(* Logix 5000 project; controller SX_V040001_C001 vendor 1 type 14 code 77 rev 16.22; software revision 16.04; part 16 of 35 *)
(* tags used below, declared in another part *)
   ALL_KINDS : INT[90];
   DRIVE : INT[32];
   G_AOutput : DINT[8];
   G_DInput : DINT[3];
   G_DOutput : DINT[3];
   NOTDOS : INT[6];
   PARAMETER : INT[501];
   T_CONTR_CLFA_ACLFA : TIMER;
   T_CURRENT_AUTO : TIMER;
   T_CURRENT_CL : TIMER;
   T_DELAY_SLOW_FAST : TIMER;
   T_DELAY_SOFTSTART : TIMER;
   T_DRIVE_START_WARN : TIMER;
(* MainProgram, continued *)

ROUTINE MainDrive2Motors   (* ladder *)
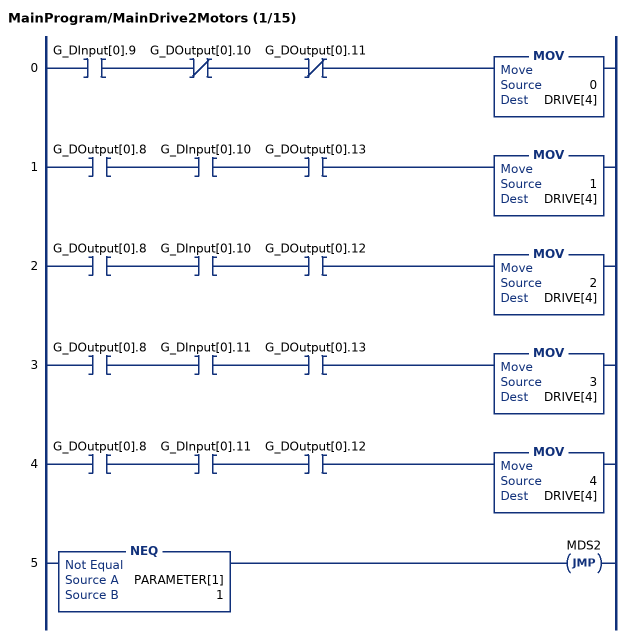
   0: XIC(G_DInput[0].9)XIO(G_DOutput[0].10)XIO(G_DOutput[0].11)MOV(0,DRIVE[4]);
   1: XIC(G_DOutput[0].8)XIC(G_DInput[0].10)XIC(G_DOutput[0].13)MOV(1,DRIVE[4]);
   2: XIC(G_DOutput[0].8)XIC(G_DInput[0].10)XIC(G_DOutput[0].12)MOV(2,DRIVE[4]);
   3: XIC(G_DOutput[0].8)XIC(G_DInput[0].11)XIC(G_DOutput[0].13)MOV(3,DRIVE[4]);
   4: XIC(G_DOutput[0].8)XIC(G_DInput[0].11)XIC(G_DOutput[0].12)MOV(4,DRIVE[4]);
   5: NEQ(PARAMETER[1],1)JMP(MDS2);
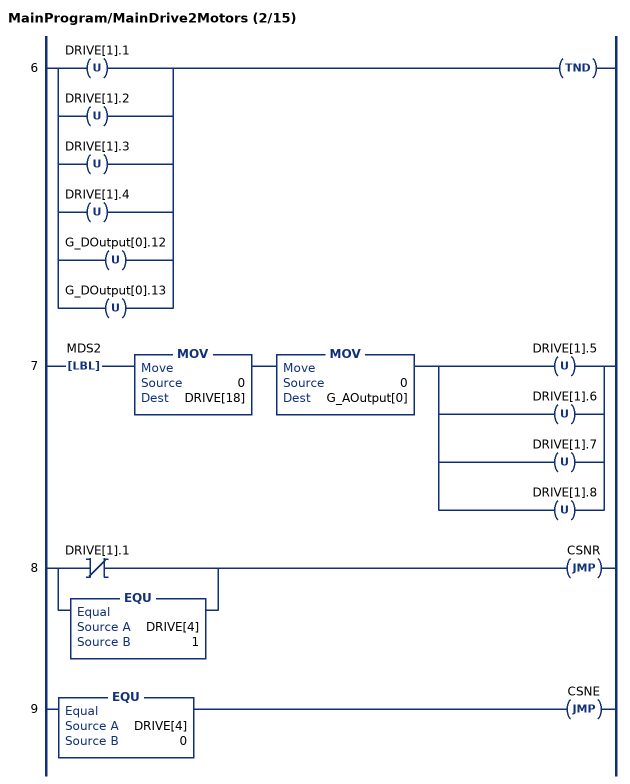
   6: [OTU(DRIVE[1].1) ,OTU(DRIVE[1].2) ,OTU(DRIVE[1].3) ,OTU(DRIVE[1].4) ,OTU(G_DOutput[0].12) ,OTU(G_DOutput[0].13) ]TND();
   7: LBL(MDS2)MOV(0,DRIVE[18])MOV(0,G_AOutput[0])[OTU(DRIVE[1].5) ,OTU(DRIVE[1].6) ,OTU(DRIVE[1].7) ,OTU(DRIVE[1].8) ];
   8: [XIO(DRIVE[1].1) ,EQU(DRIVE[4],1) ]JMP(CSNR);
   9: EQU(DRIVE[4],0)JMP(CSNE);
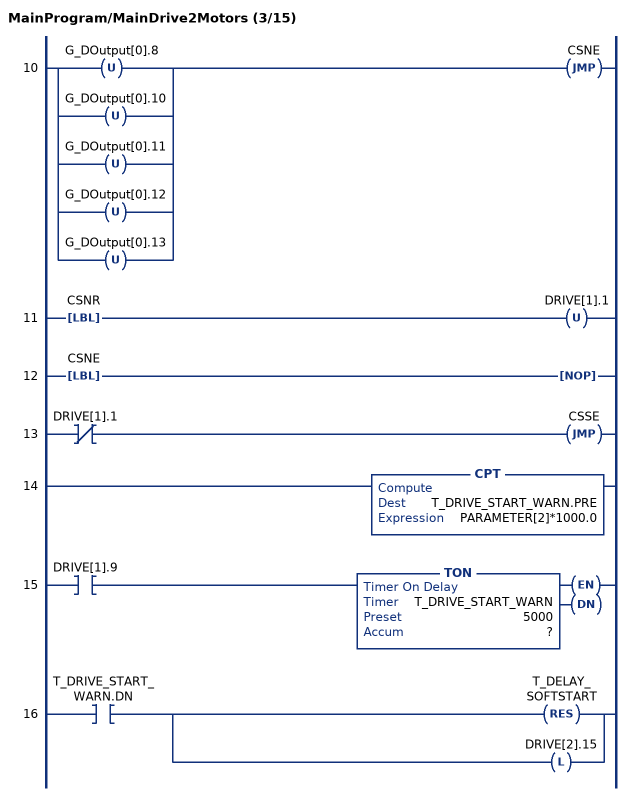
   10: [OTU(G_DOutput[0].8) ,OTU(G_DOutput[0].10) ,OTU(G_DOutput[0].11) ,OTU(G_DOutput[0].12) ,OTU(G_DOutput[0].13) ]JMP(CSNE);
   11: LBL(CSNR)OTU(DRIVE[1].1);
   12: LBL(CSNE)NOP();
   13: XIO(DRIVE[1].1)JMP(CSSE);
   14: CPT(T_DRIVE_START_WARN.PRE,PARAMETER[2]*1000.0);
   15: XIC(DRIVE[1].9)TON(T_DRIVE_START_WARN,?,?);
   16: XIC(T_DRIVE_START_WARN.DN)[RES(T_DELAY_SOFTSTART) ,OTL(DRIVE[2].15) ];
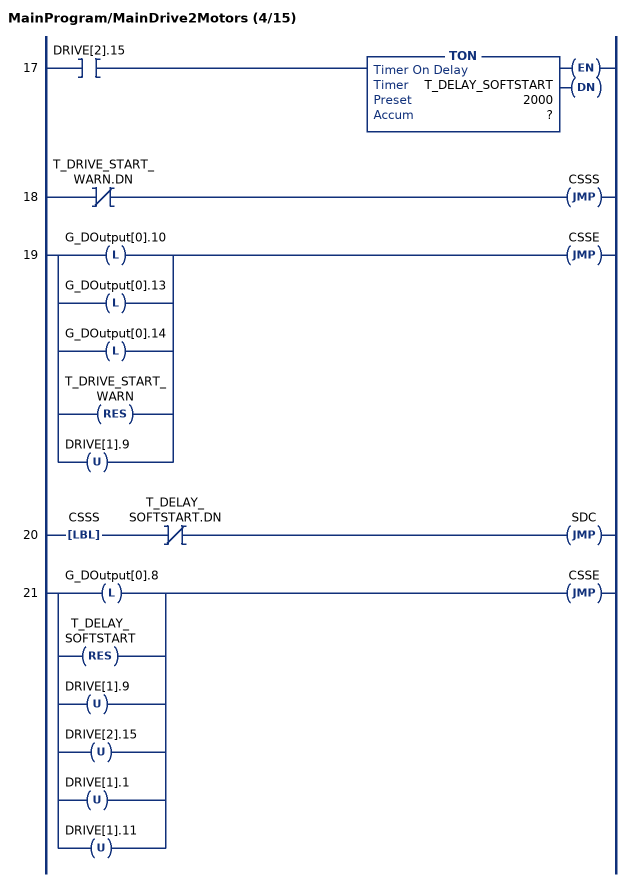
   17: XIC(DRIVE[2].15)TON(T_DELAY_SOFTSTART,?,?);
   18: XIO(T_DRIVE_START_WARN.DN)JMP(CSSS);
   19: [OTL(G_DOutput[0].10) ,OTL(G_DOutput[0].13) ,OTL(G_DOutput[0].14) ,RES(T_DRIVE_START_WARN) ,OTU(DRIVE[1].9) ]JMP(CSSE);
   20: LBL(CSSS)XIO(T_DELAY_SOFTSTART.DN)JMP(SDC);
   21: [OTL(G_DOutput[0].8) ,RES(T_DELAY_SOFTSTART) ,OTU(DRIVE[1].9) ,OTU(DRIVE[2].15) ,OTU(DRIVE[1].1) ,OTU(DRIVE[1].11) ]JMP(CSSE);
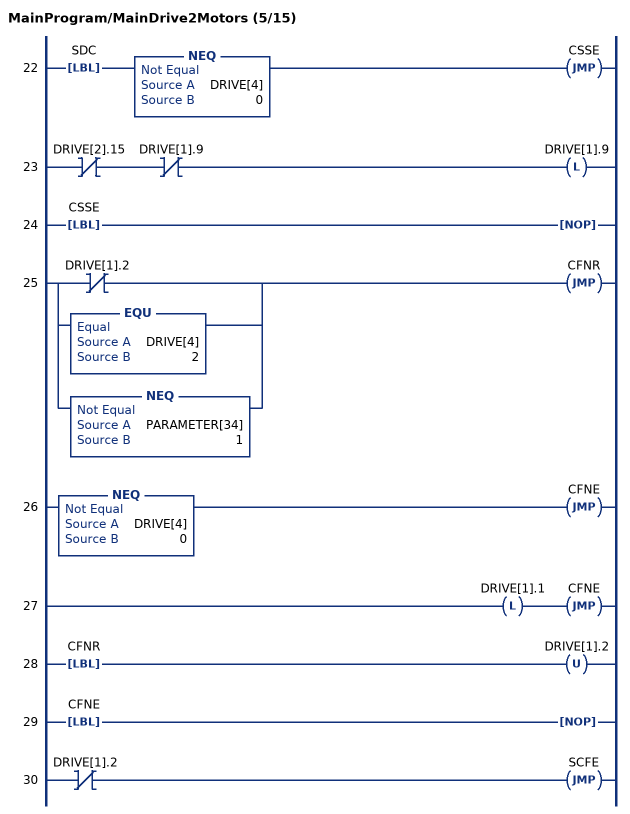
   22: LBL(SDC)NEQ(DRIVE[4],0)JMP(CSSE);
   23: XIO(DRIVE[2].15)XIO(DRIVE[1].9)OTL(DRIVE[1].9);
   24: LBL(CSSE)NOP();
   25: [XIO(DRIVE[1].2) ,EQU(DRIVE[4],2) ,NEQ(PARAMETER[34],1) ]JMP(CFNR);
   26: NEQ(DRIVE[4],0)JMP(CFNE);
   27: OTL(DRIVE[1].1)JMP(CFNE);
   28: LBL(CFNR)OTU(DRIVE[1].2);
   29: LBL(CFNE)NOP();
   30: XIO(DRIVE[1].2)JMP(SCFE);
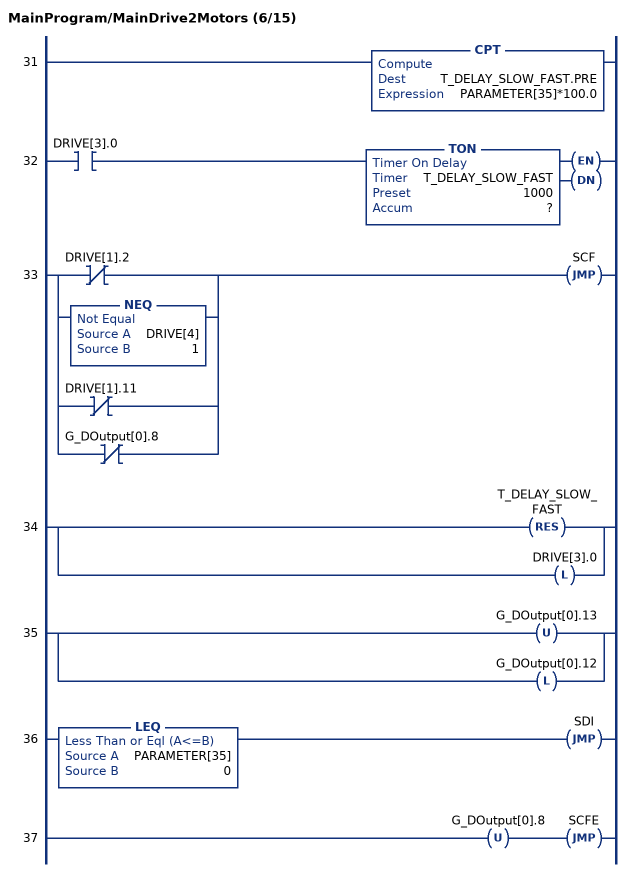
   31: CPT(T_DELAY_SLOW_FAST.PRE,PARAMETER[35]*100.0);
   32: XIC(DRIVE[3].0)TON(T_DELAY_SLOW_FAST,?,?);
   33: [XIO(DRIVE[1].2) ,NEQ(DRIVE[4],1) ,XIO(DRIVE[1].11) ,XIO(G_DOutput[0].8) ]JMP(SCF);
   34: [RES(T_DELAY_SLOW_FAST) ,OTL(DRIVE[3].0) ];
   35: [OTU(G_DOutput[0].13) ,OTL(G_DOutput[0].12) ];
   36: LEQ(PARAMETER[35],0)JMP(SDI);
   37: OTU(G_DOutput[0].8)JMP(SCFE);
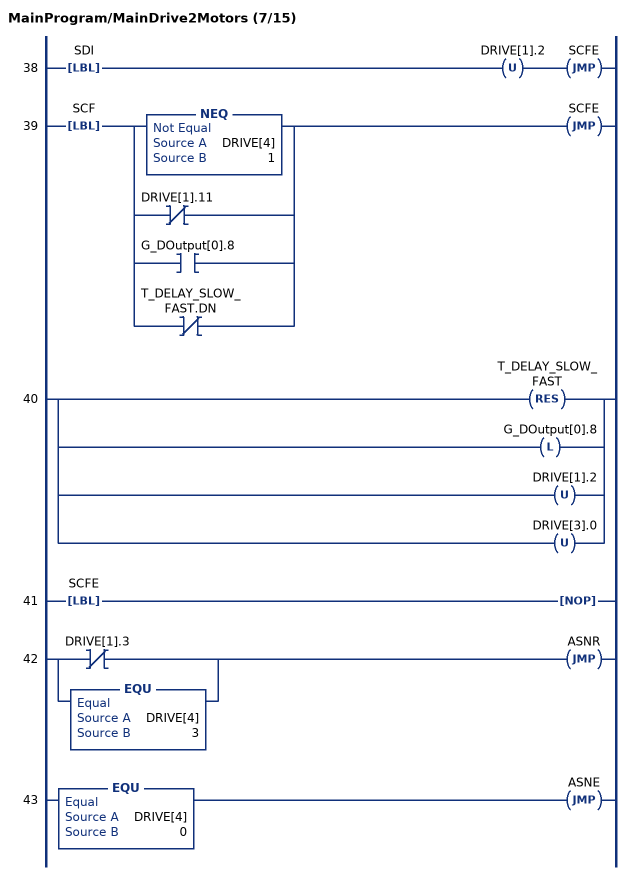
   38: LBL(SDI)OTU(DRIVE[1].2)JMP(SCFE);
   39: LBL(SCF)[NEQ(DRIVE[4],1) ,XIO(DRIVE[1].11) ,XIC(G_DOutput[0].8) ,XIO(T_DELAY_SLOW_FAST.DN) ]JMP(SCFE);
   40: [RES(T_DELAY_SLOW_FAST) ,OTL(G_DOutput[0].8) ,OTU(DRIVE[1].2) ,OTU(DRIVE[3].0) ];
   41: LBL(SCFE)NOP();
   42: [XIO(DRIVE[1].3) ,EQU(DRIVE[4],3) ]JMP(ASNR);
   43: EQU(DRIVE[4],0)JMP(ASNE);
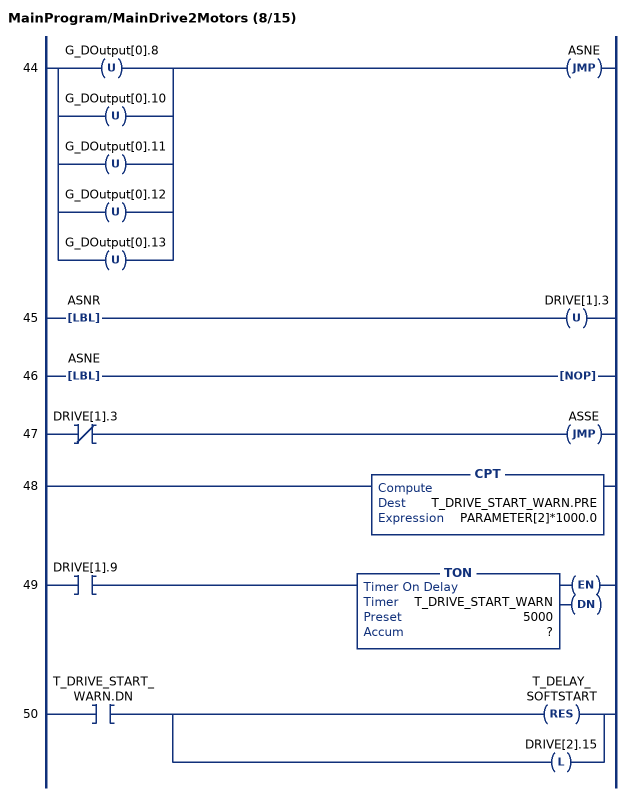
   44: [OTU(G_DOutput[0].8) ,OTU(G_DOutput[0].10) ,OTU(G_DOutput[0].11) ,OTU(G_DOutput[0].12) ,OTU(G_DOutput[0].13) ]JMP(ASNE);
   45: LBL(ASNR)OTU(DRIVE[1].3);
   46: LBL(ASNE)NOP();
   47: XIO(DRIVE[1].3)JMP(ASSE);
   48: CPT(T_DRIVE_START_WARN.PRE,PARAMETER[2]*1000.0);
   49: XIC(DRIVE[1].9)TON(T_DRIVE_START_WARN,?,?);
   50: XIC(T_DRIVE_START_WARN.DN)[RES(T_DELAY_SOFTSTART) ,OTL(DRIVE[2].15) ];
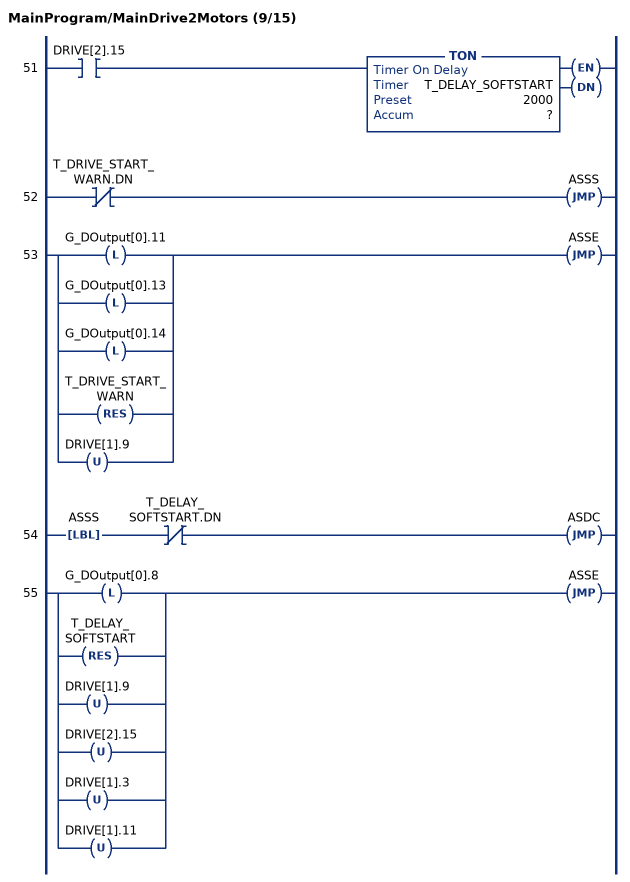
   51: XIC(DRIVE[2].15)TON(T_DELAY_SOFTSTART,?,?);
   52: XIO(T_DRIVE_START_WARN.DN)JMP(ASSS);
   53: [OTL(G_DOutput[0].11) ,OTL(G_DOutput[0].13) ,OTL(G_DOutput[0].14) ,RES(T_DRIVE_START_WARN) ,OTU(DRIVE[1].9) ]JMP(ASSE);
   54: LBL(ASSS)XIO(T_DELAY_SOFTSTART.DN)JMP(ASDC);
   55: [OTL(G_DOutput[0].8) ,RES(T_DELAY_SOFTSTART) ,OTU(DRIVE[1].9) ,OTU(DRIVE[2].15) ,OTU(DRIVE[1].3) ,OTU(DRIVE[1].11) ]JMP(ASSE);
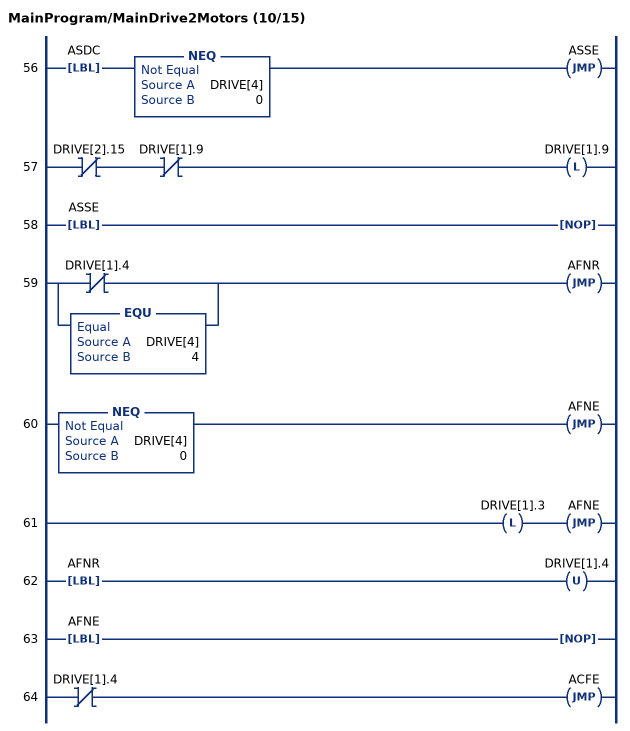
   56: LBL(ASDC)NEQ(DRIVE[4],0)JMP(ASSE);
   57: XIO(DRIVE[2].15)XIO(DRIVE[1].9)OTL(DRIVE[1].9);
   58: LBL(ASSE)NOP();
   59: [XIO(DRIVE[1].4) ,EQU(DRIVE[4],4) ]JMP(AFNR);
   60: NEQ(DRIVE[4],0)JMP(AFNE);
   61: OTL(DRIVE[1].3)JMP(AFNE);
   62: LBL(AFNR)OTU(DRIVE[1].4);
   63: LBL(AFNE)NOP();
   64: XIO(DRIVE[1].4)JMP(ACFE);
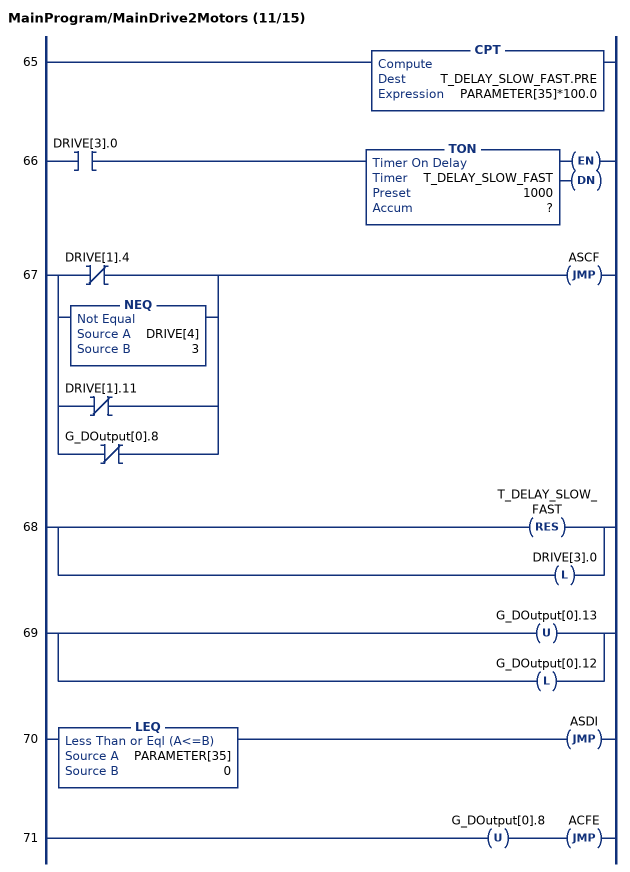
   65: CPT(T_DELAY_SLOW_FAST.PRE,PARAMETER[35]*100.0);
   66: XIC(DRIVE[3].0)TON(T_DELAY_SLOW_FAST,?,?);
   67: [XIO(DRIVE[1].4) ,NEQ(DRIVE[4],3) ,XIO(DRIVE[1].11) ,XIO(G_DOutput[0].8) ]JMP(ASCF);
   68: [RES(T_DELAY_SLOW_FAST) ,OTL(DRIVE[3].0) ];
   69: [OTU(G_DOutput[0].13) ,OTL(G_DOutput[0].12) ];
   70: LEQ(PARAMETER[35],0)JMP(ASDI);
   71: OTU(G_DOutput[0].8)JMP(ACFE);
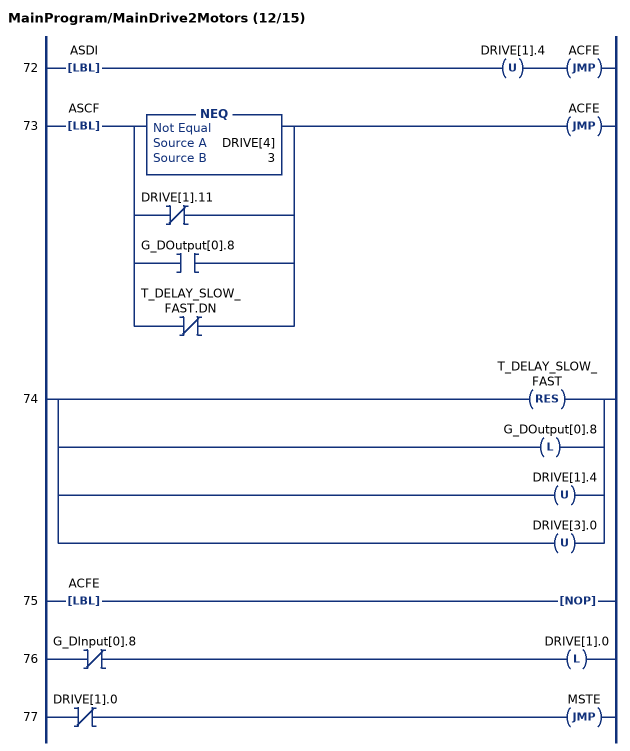
   72: LBL(ASDI)OTU(DRIVE[1].4)JMP(ACFE);
   73: LBL(ASCF)[NEQ(DRIVE[4],3) ,XIO(DRIVE[1].11) ,XIC(G_DOutput[0].8) ,XIO(T_DELAY_SLOW_FAST.DN) ]JMP(ACFE);
   74: [RES(T_DELAY_SLOW_FAST) ,OTL(G_DOutput[0].8) ,OTU(DRIVE[1].4) ,OTU(DRIVE[3].0) ];
   75: LBL(ACFE)NOP();
   76: XIO(G_DInput[0].8)OTL(DRIVE[1].0);
   77: XIO(DRIVE[1].0)JMP(MSTE);
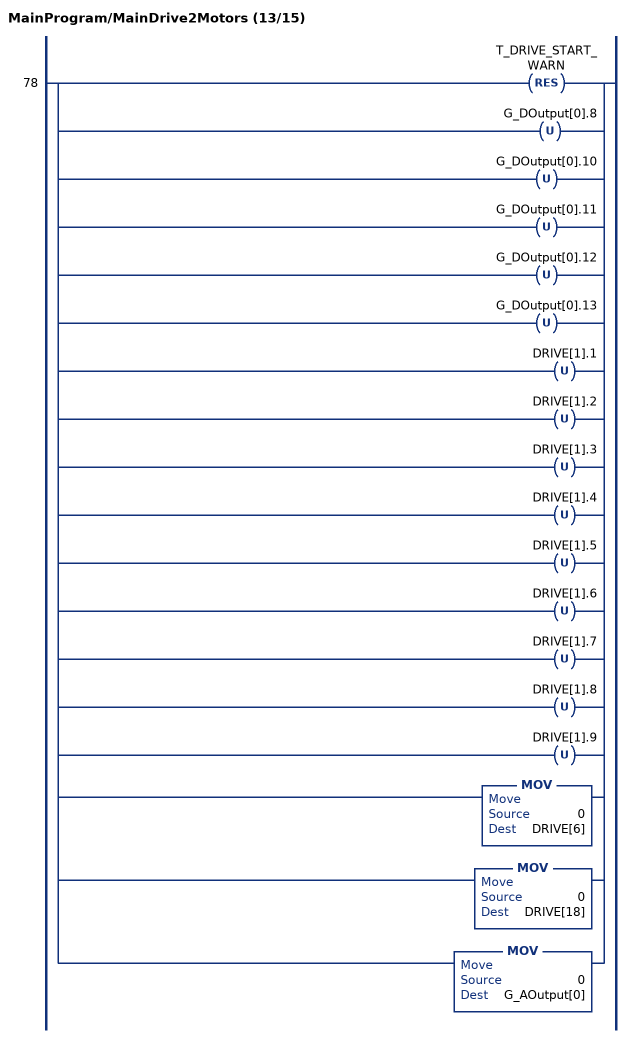
   78: [RES(T_DRIVE_START_WARN) ,OTU(G_DOutput[0].8) ,OTU(G_DOutput[0].10) ,OTU(G_DOutput[0].11) ,OTU(G_DOutput[0].12) ,OTU(G_DOutput[0].13) ,OTU(DRIVE[1].1) ,OTU(DRIVE[1].2) ,OTU(DRIVE[1].3) ,OTU(DRIVE[1].4) ,OTU(DRIVE[1].5) ,OTU(DRIVE[1].6) ,OTU(DRIVE[1].7) ,OTU(DRIVE[1].8) ,OTU(DRIVE[1].9) ,MOV(0,DRIVE[6]) ,MOV(0,DRIVE[18]) ,MOV(0,G_AOutput[0]) ];
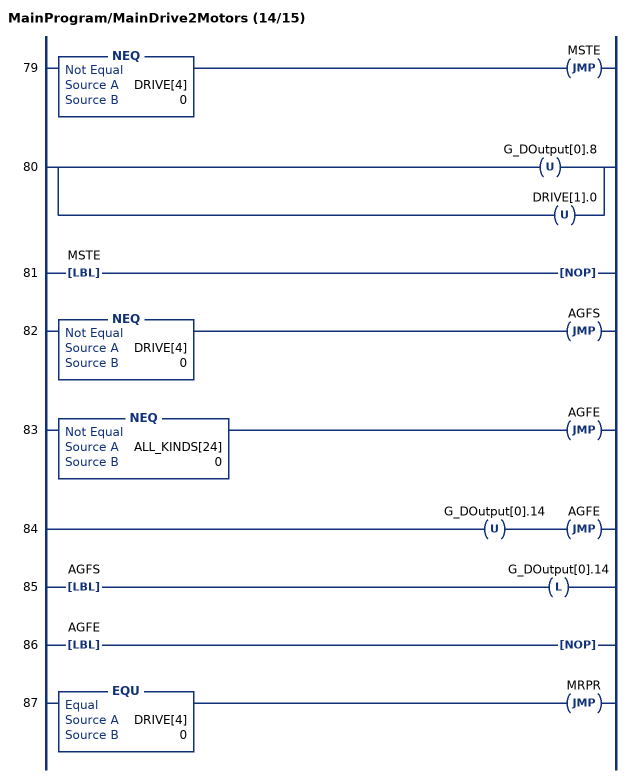
   79: NEQ(DRIVE[4],0)JMP(MSTE);
   80: [OTU(G_DOutput[0].8) ,OTU(DRIVE[1].0) ];
   81: LBL(MSTE)NOP();
   82: NEQ(DRIVE[4],0)JMP(AGFS);
   83: NEQ(ALL_KINDS[24],0)JMP(AGFE);
   84: OTU(G_DOutput[0].14)JMP(AGFE);
   85: LBL(AGFS)OTL(G_DOutput[0].14);
   86: LBL(AGFE)NOP();
   87: EQU(DRIVE[4],0)JMP(MRPR);
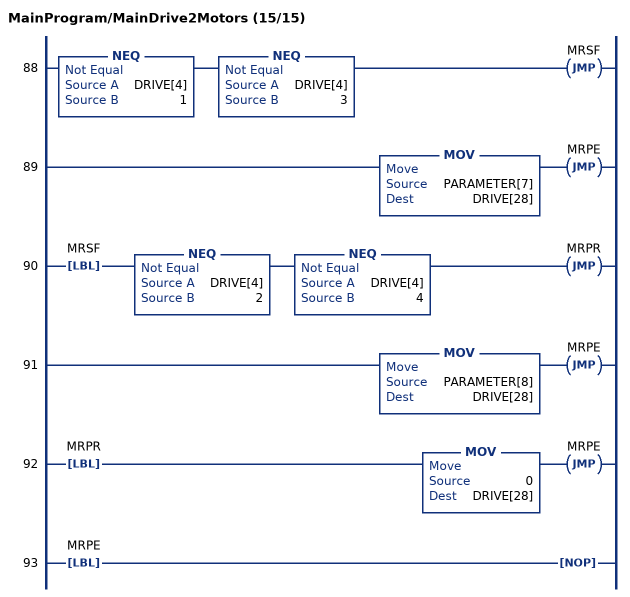
   88: NEQ(DRIVE[4],1)NEQ(DRIVE[4],3)JMP(MRSF);
   89: MOV(PARAMETER[7],DRIVE[28])JMP(MRPE);
   90: LBL(MRSF)NEQ(DRIVE[4],2)NEQ(DRIVE[4],4)JMP(MRPR);
   91: MOV(PARAMETER[8],DRIVE[28])JMP(MRPE);
   92: LBL(MRPR)MOV(0,DRIVE[28])JMP(MRPE);
   93: LBL(MRPE)NOP();
END_ROUTINE

ROUTINE MainDriveCurrent   (* ladder *)
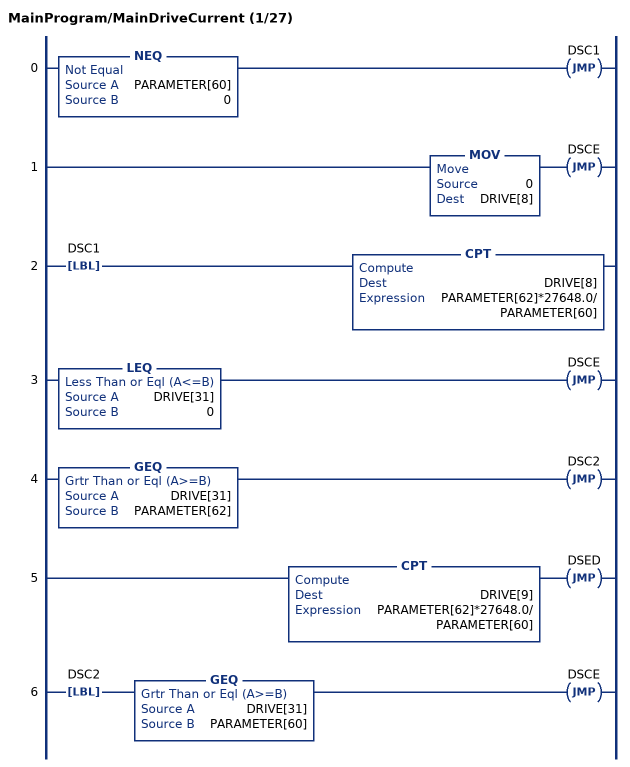
   0: NEQ(PARAMETER[60],0)JMP(DSC1);
   1: MOV(0,DRIVE[8])JMP(DSCE);
   2: LBL(DSC1)CPT(DRIVE[8],PARAMETER[62]*27648.0/PARAMETER[60]);
   3: LEQ(DRIVE[31],0)JMP(DSCE);
   4: GEQ(DRIVE[31],PARAMETER[62])JMP(DSC2);
   5: CPT(DRIVE[9],PARAMETER[62]*27648.0/PARAMETER[60])JMP(DSED);
   6: LBL(DSC2)GEQ(DRIVE[31],PARAMETER[60])JMP(DSCE);
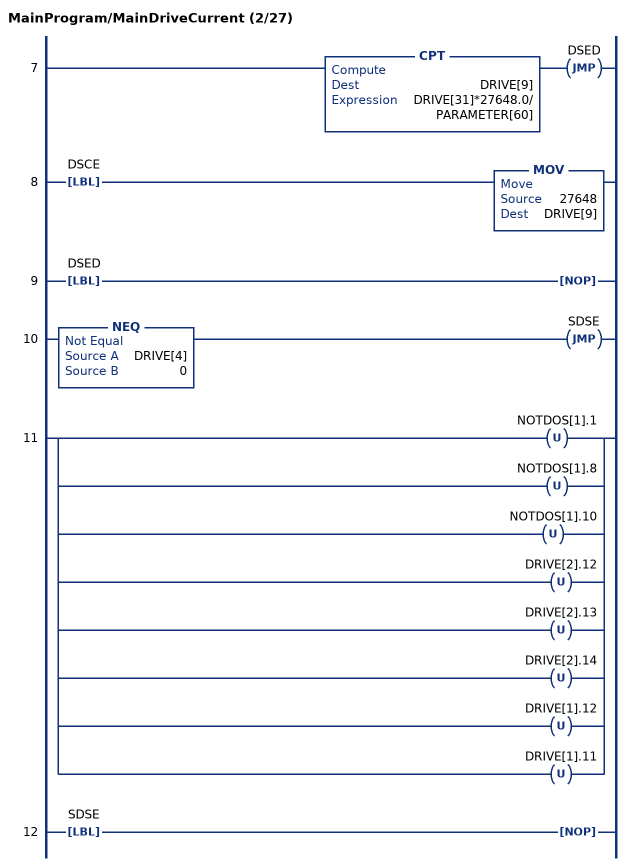
   7: CPT(DRIVE[9],DRIVE[31]*27648.0/PARAMETER[60])JMP(DSED);
   8: LBL(DSCE)MOV(27648,DRIVE[9]);
   9: LBL(DSED)NOP();
   10: NEQ(DRIVE[4],0)JMP(SDSE);
   11: [OTU(NOTDOS[1].1) ,OTU(NOTDOS[1].8) ,OTU(NOTDOS[1].10) ,OTU(DRIVE[2].12) ,OTU(DRIVE[2].13) ,OTU(DRIVE[2].14) ,OTU(DRIVE[1].12) ,OTU(DRIVE[1].11) ];
   12: LBL(SDSE)NOP();
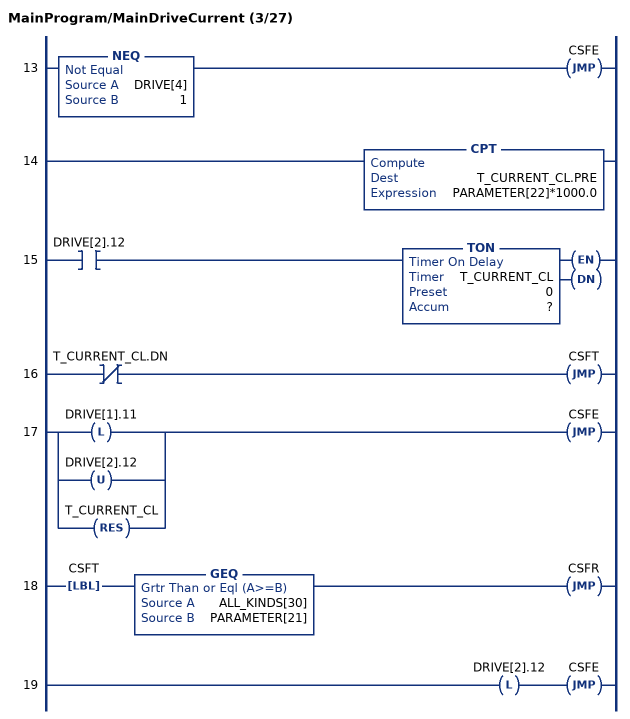
   13: NEQ(DRIVE[4],1)JMP(CSFE);
   14: CPT(T_CURRENT_CL.PRE,PARAMETER[22]*1000.0);
   15: XIC(DRIVE[2].12)TON(T_CURRENT_CL,?,?);
   16: XIO(T_CURRENT_CL.DN)JMP(CSFT);
   17: [OTL(DRIVE[1].11) ,OTU(DRIVE[2].12) ,RES(T_CURRENT_CL) ]JMP(CSFE);
   18: LBL(CSFT)GEQ(ALL_KINDS[30],PARAMETER[21])JMP(CSFR);
   19: OTL(DRIVE[2].12)JMP(CSFE);
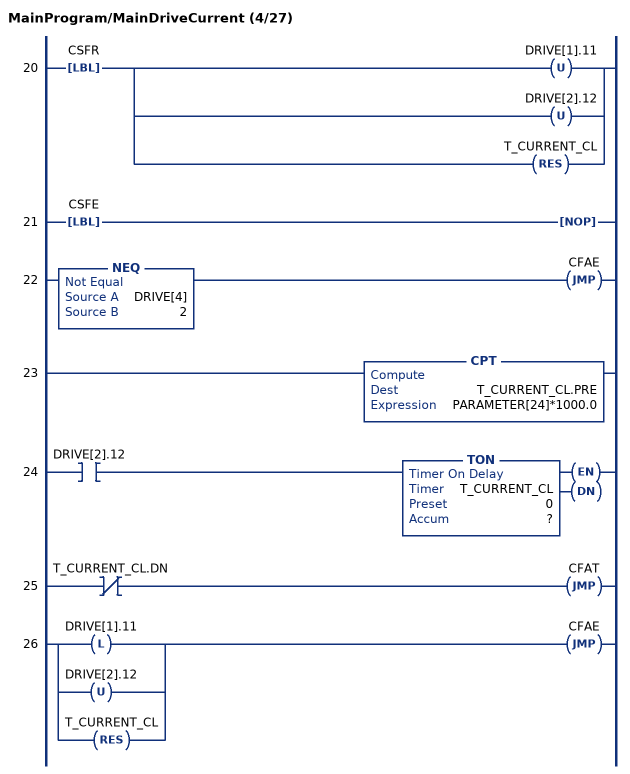
   20: LBL(CSFR)[OTU(DRIVE[1].11) ,OTU(DRIVE[2].12) ,RES(T_CURRENT_CL) ];
   21: LBL(CSFE)NOP();
   22: NEQ(DRIVE[4],2)JMP(CFAE);
   23: CPT(T_CURRENT_CL.PRE,PARAMETER[24]*1000.0);
   24: XIC(DRIVE[2].12)TON(T_CURRENT_CL,?,?);
   25: XIO(T_CURRENT_CL.DN)JMP(CFAT);
   26: [OTL(DRIVE[1].11) ,OTU(DRIVE[2].12) ,RES(T_CURRENT_CL) ]JMP(CFAE);
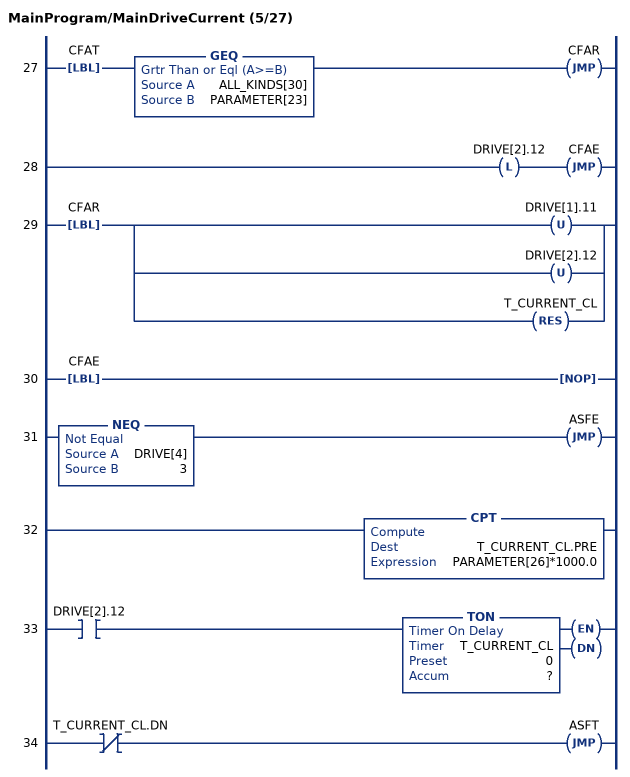
   27: LBL(CFAT)GEQ(ALL_KINDS[30],PARAMETER[23])JMP(CFAR);
   28: OTL(DRIVE[2].12)JMP(CFAE);
   29: LBL(CFAR)[OTU(DRIVE[1].11) ,OTU(DRIVE[2].12) ,RES(T_CURRENT_CL) ];
   30: LBL(CFAE)NOP();
   31: NEQ(DRIVE[4],3)JMP(ASFE);
   32: CPT(T_CURRENT_CL.PRE,PARAMETER[26]*1000.0);
   33: XIC(DRIVE[2].12)TON(T_CURRENT_CL,?,?);
   34: XIO(T_CURRENT_CL.DN)JMP(ASFT);
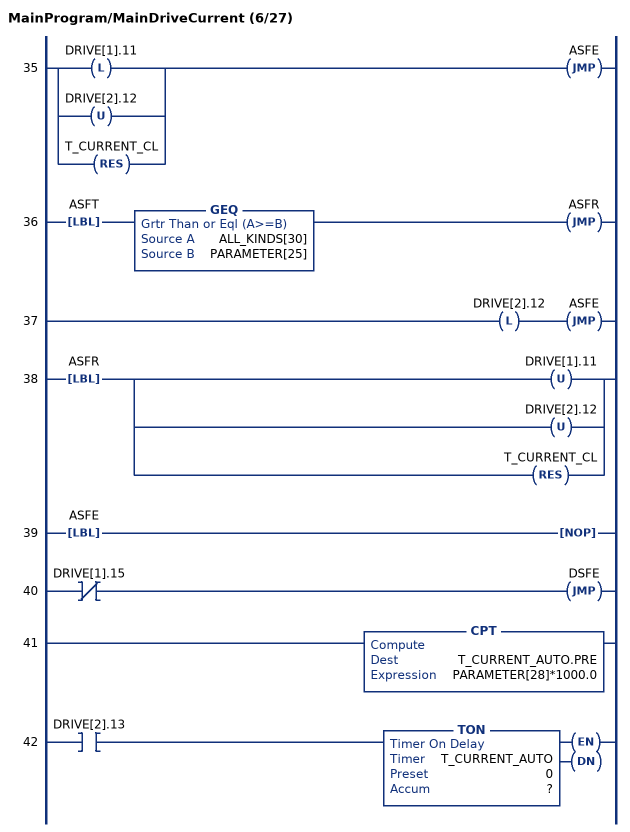
   35: [OTL(DRIVE[1].11) ,OTU(DRIVE[2].12) ,RES(T_CURRENT_CL) ]JMP(ASFE);
   36: LBL(ASFT)GEQ(ALL_KINDS[30],PARAMETER[25])JMP(ASFR);
   37: OTL(DRIVE[2].12)JMP(ASFE);
   38: LBL(ASFR)[OTU(DRIVE[1].11) ,OTU(DRIVE[2].12) ,RES(T_CURRENT_CL) ];
   39: LBL(ASFE)NOP();
   40: XIO(DRIVE[1].15)JMP(DSFE);
   41: CPT(T_CURRENT_AUTO.PRE,PARAMETER[28]*1000.0);
   42: XIC(DRIVE[2].13)TON(T_CURRENT_AUTO,?,?);
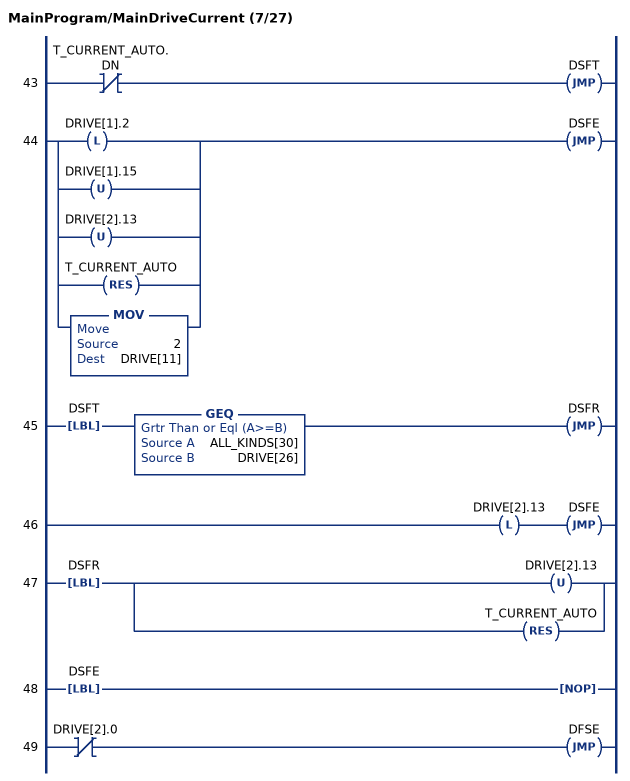
   43: XIO(T_CURRENT_AUTO.DN)JMP(DSFT);
   44: [OTL(DRIVE[1].2) ,OTU(DRIVE[1].15) ,OTU(DRIVE[2].13) ,RES(T_CURRENT_AUTO) ,MOV(2,DRIVE[11]) ]JMP(DSFE);
   45: LBL(DSFT)GEQ(ALL_KINDS[30],DRIVE[26])JMP(DSFR);
   46: OTL(DRIVE[2].13)JMP(DSFE);
   47: LBL(DSFR)[OTU(DRIVE[2].13) ,RES(T_CURRENT_AUTO) ];
   48: LBL(DSFE)NOP();
   49: XIO(DRIVE[2].0)JMP(DFSE);
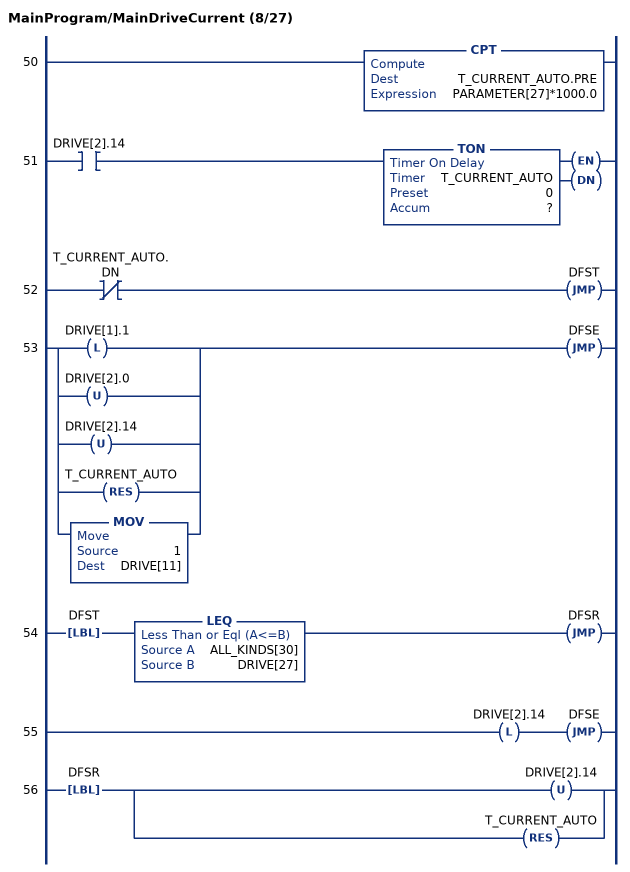
   50: CPT(T_CURRENT_AUTO.PRE,PARAMETER[27]*1000.0);
   51: XIC(DRIVE[2].14)TON(T_CURRENT_AUTO,?,?);
   52: XIO(T_CURRENT_AUTO.DN)JMP(DFST);
   53: [OTL(DRIVE[1].1) ,OTU(DRIVE[2].0) ,OTU(DRIVE[2].14) ,RES(T_CURRENT_AUTO) ,MOV(1,DRIVE[11]) ]JMP(DFSE);
   54: LBL(DFST)LEQ(ALL_KINDS[30],DRIVE[27])JMP(DFSR);
   55: OTL(DRIVE[2].14)JMP(DFSE);
   56: LBL(DFSR)[OTU(DRIVE[2].14) ,RES(T_CURRENT_AUTO) ];
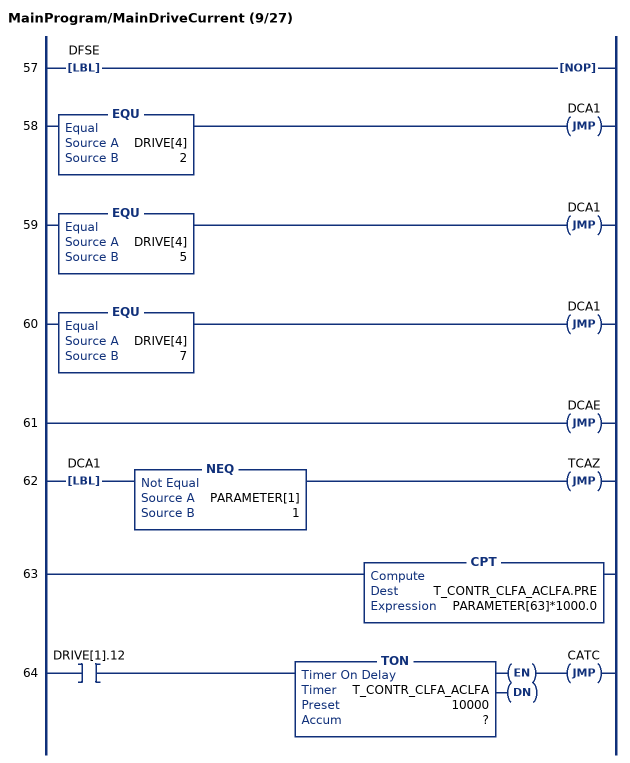
   57: LBL(DFSE)NOP();
   58: EQU(DRIVE[4],2)JMP(DCA1);
   59: EQU(DRIVE[4],5)JMP(DCA1);
   60: EQU(DRIVE[4],7)JMP(DCA1);
   61: JMP(DCAE);
   62: LBL(DCA1)NEQ(PARAMETER[1],1)JMP(TCAZ);
   63: CPT(T_CONTR_CLFA_ACLFA.PRE,PARAMETER[63]*1000.0);
   64: XIC(DRIVE[1].12)TON(T_CONTR_CLFA_ACLFA,?,?)JMP(CATC);
